FUNCTION_BLOCK LedLogic
VAR_INPUT
END_VAR
VAR_OUTPUT
END_VAR
VAR
END_VAR

END_FUNCTION_BLOCK

(* stored: Version 1.1.0.1, ProductVersion 3.1.4024.14
   POU LedLogic: Id {8faa0091-5f1c-4918-9cd9-098492844bdf}, SpecialFunc None *)
